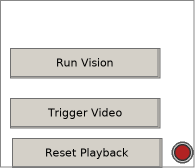
VISUALIZATION V_Main  // 195x168
    Button (10,48 150x30), "Run Vision"
        toggle MAIN.Camera1.RunVision
    Button (10,98 150x30), "Trigger Video"
        toggle MAIN.TriggerEvent
    Button (12,138 150x30), "Reset Playback"
        tap MAIN.Playback._Reset
    Lamp1 (170,140 25x25), variable: MAIN.Playback._Error, style: Lamp-Lamp1-Red
END_VISUALIZATION

(* stored: Version 1.1.0.1, ProductVersion 3.1.4024.13
   Visu V_Main: Id {48cf825d-6f3d-4f02-92db-e2c8f42e68b5} *)
